// TIA Portal V17 program export: 3 tag tables, 41 data types, 3 data blocks, 7 code blocks (in call order from the OBs), 4 instance data blocks

VAR_GLOBAL   // PLC tag table "Constants"
END_VAR
VAR_GLOBAL CONSTANT   // user constants
   LASERCOMM_LDD_ARRAY_SIZE : Int := 100;   // Size of LDD Array Data Sizes. This is for Results, DDO and Weld Mask. Tied to the number of jobs in the LDD Sequence.
   LASERCOMM_NUMBER_OF_LASERS : Int := 1;   // Number of Lasers systems on Cell
   LASERCOMM_REF_PLANE : DInt := 12345;   // LDD Reference Plane Position
END_VAR

VAR_GLOBAL   // PLC tag table "Default tag table"
   Start_Seq AT %M0.0 : Bool;
   Rob_Reset_1 AT %M0.1 : Bool;
   Rob_Reset_2 AT %M0.2 : Bool;
   RA_CC_1 AT %M0.3 : Bool;
END_VAR
VAR_GLOBAL CONSTANT   // user constants
   GRP_JOB_NAME_SIZE : Int := 50;   // String site group and job name / String Größe Gruppen- und Jobnamen
   MAX_CNT_GRP_OVR_ENTRIES : DInt := 100;   // Maximum number of groups in the group overview / Maximale Anzahl Gruppen in der Gruppen-Übersicht
   MAX_CNT_MTN_OVR_ENTRIES : DInt := 150;   // Maximum number of motions in the motion overview / Maximale Anzahl Motions in der Motion-Übersicht
END_VAR

VAR_GLOBAL   // PLC tag table "Standard IO"
   iScanner1 AT %I0.0 : "Scanner_Inputs";
   oScanner1 AT %Q0.0 : "Scanner_Outputs";
   iLaser1 AT %I48.0 : "YLS_Inputs";
   oLaser1 AT %Q32.0 : "YLS_Outputs";
END_VAR

TYPE "typeAnalogSensorUniversalLimits"
// stored: IsFailsafeCompliant false
   STRUCT
      minPosition { ExternalAccessible := 'False'; ExternalVisible := 'False'; ExternalWritable := 'False'} : Array[1..8] of LReal;   // minimale Position / Minimum position
      maxPosition { ExternalAccessible := 'False'; ExternalVisible := 'False'; ExternalWritable := 'False'} : Array[1..8] of LReal;   // maximale Position / Maximum position
   END_STRUCT;
END_TYPE

TYPE "typeAnalogSensorUniversalPositions"
// stored: IsFailsafeCompliant false
   STRUCT
      inPosition { ExternalAccessible := 'False'; ExternalVisible := 'False'; ExternalWritable := 'False'} : Array[1..8] of Bool;   // in Position / In position
   END_STRUCT;
END_TYPE

TYPE "typeCaCgFg"
TITLE = Group / Gruppe
// Gruppe [V 01.09 | Kernel_V2]
// stored: IsFailsafeCompliant false
   STRUCT
      info { ExternalAccessible := 'False'; ExternalVisible := 'False'; ExternalWritable := 'False'} : Struct   // Info / Information
         "name" { ExternalAccessible := 'False'; ExternalVisible := 'False'; ExternalWritable := 'False'} : WString["GRP_JOB_NAME_SIZE"];   // Bezeichnung / Designation
         idString { ExternalAccessible := 'False'; ExternalVisible := 'False'; ExternalWritable := 'False'} : WString["GRP_JOB_NAME_SIZE"];   // ID-Bezeichnung als String (originaler Name des Gruppen-DB)
         groupType { ExternalAccessible := 'False'; ExternalVisible := 'False'; ExternalWritable := 'False'} : Int;   // Typ (1= CA | 2= CG | 3= FG) / Type (1 = CA | 2 = CG | 3 = FG)
         dbAdress { ExternalAccessible := 'False'; ExternalVisible := 'False'; ExternalWritable := 'False'} : DB_ANY;   // DB-Adresse der Gruppeschnittstelle (typeCaCgFg) / DB address of group interface (typeCaCgFg)
         panel { ExternalAccessible := 'False'; ExternalVisible := 'False'; ExternalWritable := 'False'} : Struct   // Panel
            assignment { ExternalAccessible := 'False'; ExternalVisible := 'False'; ExternalWritable := 'False'} : Int;   // Hmi Panel Zuweisung (Panel-Index aus HMI Lite) / HMI panel assignment (panel index from HMI Lite)
            memoryIndex { ExternalAccessible := 'False'; ExternalVisible := 'False'; ExternalWritable := 'False'} : Int;   // Speicherplatz Index Panel-Bild / Memory index panel screen
         END_STRUCT;
         parentGroup { ExternalAccessible := 'False'; ExternalVisible := 'False'; ExternalWritable := 'False'} : Struct   // Übergeordnete Gruppe / Superordinate group
            groupType { ExternalAccessible := 'False'; ExternalVisible := 'False'; ExternalWritable := 'False'} : Int;   // Übergeordnete Gruppe: Typ (1= CA | 2= CG | 3= FG) / Superordinate group: Type (1 = CA | 2 = CG | 3 = FG)
            "name" { ExternalAccessible := 'False'; ExternalVisible := 'False'; ExternalWritable := 'False'} : WString["GRP_JOB_NAME_SIZE"];   // Übergeordnete Gruppe: Bezeichnung / Superordinate group: Designation
            dbAdress { ExternalAccessible := 'False'; ExternalVisible := 'False'; ExternalWritable := 'False'} : DB_ANY;   // Übergeordnete Gruppe: DB-Adresse der Gruppeschnittstelle (typeCaCgFg) / Superordinate group: DB address of group interface (typeCaCgFg)
         END_STRUCT;
         groupOvrv { ExternalAccessible := 'False'; ExternalVisible := 'False'; ExternalWritable := 'False'} : Struct   // Gruppenübersichtstabelle: ... / Group overview table: ...
            groupOvrvAdress { ExternalAccessible := 'False'; ExternalVisible := 'False'; ExternalWritable := 'False'} : DB_ANY;   // Gruppenübersichtstabelle: Adresse auf Gruppenübersichts-DB (typeGroupOvrvList) / Group overview table: address on group overview DB (typeGroupOvrvList)
            listedIndex { ExternalAccessible := 'False'; ExternalVisible := 'False'; ExternalWritable := 'False'} : DInt := -1;   // Gruppenübersichtstabelle: Index der Gruppe im Gruppenübersichts-DB / Group overview table: group index in group overview DB
         END_STRUCT;
         motionOvrv { ExternalAccessible := 'False'; ExternalVisible := 'False'; ExternalWritable := 'False'} : Struct   // Motion-Übersichtstabelle: ... (Wird nur in einer FG beschrieben!) / Motion overview table: ... (only described in one FG!)
            enabled { ExternalAccessible := 'False'; ExternalVisible := 'False'; ExternalWritable := 'False'} : Bool;   // Motion-Übersichtstabelle: Freigeschaltet / Motion overview: activated
            motionOvrvAdress { ExternalAccessible := 'False'; ExternalVisible := 'False'; ExternalWritable := 'False'} : DB_ANY;   // Motion-Übersichtstabelle: Adresse auf Motion-Übersichts-DB (typeMotionOvrvList) / Motion overview table: address on motion overview DB (typeMotionOvrvList)
         END_STRUCT;
      END_STRUCT;
      groupModes { ExternalAccessible := 'False'; ExternalVisible := 'False'; ExternalWritable := 'False'} : Struct   // Gruppen Modus / Station mode <ToBeDone: determine symbol> / Group mode
         activation { ExternalAccessible := 'False'; ExternalVisible := 'False'; ExternalWritable := 'False'} : Struct   // Gruppen-Aktivierung / Group activation
            deactivate { ExternalAccessible := 'False'; ExternalVisible := 'False'; ExternalWritable := 'False'} : Bool;   // Gruppe deaktivieren (S) / Deactivate group (S)
            activate { ExternalAccessible := 'False'; ExternalVisible := 'False'; ExternalWritable := 'False'} : Bool;   // Gruppe aktivieren (S) / Activate group (S)
            isDeactived { ExternalAccessible := 'False'; ExternalVisible := 'False'; ExternalWritable := 'False'} : Bool;   // Gruppe ist deaktiviert / Group deactivated
         END_STRUCT;
         interlinkedMode { ExternalAccessible := 'False'; ExternalVisible := 'False'; ExternalWritable := 'False'} : Struct   // Verketteter Betrieb / Interlinked mode
            select { ExternalAccessible := 'False'; ExternalVisible := 'False'; ExternalWritable := 'False'} : Bool;   // Anwahl verketteter Betrieb (S) / Selection of interlinked mode (S)
            deselect { ExternalAccessible := 'False'; ExternalVisible := 'False'; ExternalWritable := 'False'} : Bool;   // Abwahl verketteter Betrieb (S) / Deselection of interlinked mode (S)
            isActive { ExternalAccessible := 'False'; ExternalVisible := 'False'; ExternalWritable := 'False'} : Bool;   // Verketteter Betrieb ist aktiv / Interlinked mode active
         END_STRUCT;
      END_STRUCT;
      enable { ExternalAccessible := 'False'; ExternalVisible := 'False'; ExternalWritable := 'False'} : Struct   // Freigaben / Enables
         hardware { ExternalAccessible := 'False'; ExternalVisible := 'False'; ExternalWritable := 'False'} : Bool;   // Freigabe Hardware betriebsbereit / Enable hardware ready for operation
         safety { ExternalAccessible := 'False'; ExternalVisible := 'False'; ExternalWritable := 'False'} : Bool;   // Freigabe Schutzbereich Bewegungsfreigabe / Enable guarded area movement enable
         enterSafeArea { ExternalAccessible := 'False'; ExternalVisible := 'False'; ExternalWritable := 'False'} : Struct   // Freigabe Zugang Schutzbereich / Enable for access guarded area
            isEnabled { ExternalAccessible := 'False'; ExternalVisible := 'False'; ExternalWritable := 'False'} : Bool;   // Zugang zum Schutzbereich ist freigegeben / Access to guarded area enabled
            disable { ExternalAccessible := 'False'; ExternalVisible := 'False'; ExternalWritable := 'False'} : Bool;   // Freigabe Zugnag Schutzbereich sperren (S) / Enable for lock access guarded area (S)
            disableSelected { ExternalAccessible := 'False'; ExternalVisible := 'False'; ExternalWritable := 'False'} : Bool;   // Freigabe Zugnag Schutzbereich sperren ist Angewählt / Enable for lock access guarded area is selected
            request { ExternalAccessible := 'False'; ExternalVisible := 'False'; ExternalWritable := 'False'} : Bool;   // Freigabe Zugang Schutzbereich anfordern (S) / Request enable for access guarded area (S)
            isRequested { ExternalAccessible := 'False'; ExternalVisible := 'False'; ExternalWritable := 'False'} : Bool;   // Freigabe Zugang Schutzbereich ist anfordert / Enable for access guarded area is requested
            operatorGuidance { ExternalAccessible := 'False'; ExternalVisible := 'False'; ExternalWritable := 'False'} : Struct   // Freigabe Zugang Schutzbereich Bedienerführung / Operator guidance guarded area access enable
               select { ExternalAccessible := 'False'; ExternalVisible := 'False'; ExternalWritable := 'False'} : Bool;   // Freigabe Zugang Schutzbereich Bedienerführung Anwahl (S) / Enable for access guarded area operator guidance selection (S)
               isSelected { ExternalAccessible := 'False'; ExternalVisible := 'False'; ExternalWritable := 'False'} : Bool;   // Freigabe Zugang Schutzbereich Bedienerführung angewählt / Operator guidance guarded area access enable selected
            END_STRUCT;
         END_STRUCT;
      END_STRUCT;
      baseFunction { ExternalAccessible := 'False'; ExternalVisible := 'False'; ExternalWritable := 'False'} : Struct   // Grundfunktionen / Basic functions
         homePos { ExternalAccessible := 'False'; ExternalVisible := 'False'; ExternalWritable := 'False'} : Struct   // Grundfunktion: Grundstellung / Basic function: home position
            select { ExternalAccessible := 'False'; ExternalVisible := 'False'; ExternalWritable := 'False'} : Bool;   // Grundfunktion: Anwahl "Zur Grundstellung" (S) / Basic function: selection "To home position" (S)
            isSelected { ExternalAccessible := 'False'; ExternalVisible := 'False'; ExternalWritable := 'False'} : Bool;   // Grundfunktion: "Zur Grundstellung" angewählt / Basic function: "To home position" selected
            isPending { ExternalAccessible := 'False'; ExternalVisible := 'False'; ExternalWritable := 'False'} : Bool;   // Grundfunktion: "Zur Grundstellung" steht an (aktiv oder gestoppt) / Basic function: "To home position" pending (active or stopped)
            inExecution { ExternalAccessible := 'False'; ExternalVisible := 'False'; ExternalWritable := 'False'} : Bool;   // Grundfunktion: "Zur Grundstellung" aktiv / Basic function: "To home position" active
            inExecutionPulse { ExternalAccessible := 'False'; ExternalVisible := 'False'; ExternalWritable := 'False'} : Bool;   // Grundfunktion: "Zur Grundstellung" aktiv Impuls / To home position active impulse / Basic function: "To home pos." active impulse
            inState { ExternalAccessible := 'False'; ExternalVisible := 'False'; ExternalWritable := 'False'} : Bool;   // Grundfunktion: In Grundstellung / Basic function: in home position
            display { ExternalAccessible := 'False'; ExternalVisible := 'False'; ExternalWritable := 'False'} : Bool;   // Grundfunktion: Grundstellung Anzeige / Basic function: home position display
            operatorGuidance { ExternalAccessible := 'False'; ExternalVisible := 'False'; ExternalWritable := 'False'} : Struct   // Grundfunktion: Bedienerfürhung / Basic function: Operator guidance
               select { ExternalAccessible := 'False'; ExternalVisible := 'False'; ExternalWritable := 'False'} : Bool;   // Grundfunktion: Bedienerfürhung Anwahl (S) / Basic function: Operator guidance selection (S)
               isSelected { ExternalAccessible := 'False'; ExternalVisible := 'False'; ExternalWritable := 'False'} : Bool;   // Grundfunktion: Bedienerfürhung Angewählt / Basic function: Operator guidance selected
            END_STRUCT;
         END_STRUCT;
         start { ExternalAccessible := 'False'; ExternalVisible := 'False'; ExternalWritable := 'False'} : Struct   // Grundfunktion: Start / Basic function: start
            select { ExternalAccessible := 'False'; ExternalVisible := 'False'; ExternalWritable := 'False'} : Bool;   // Grundfunktion: Anwah Startl (S) / Basic function: selection start (S)
            isSelected { ExternalAccessible := 'False'; ExternalVisible := 'False'; ExternalWritable := 'False'} : Bool;   // Grundfunktion: Start angewählt / Basic function: start selected
            isPending { ExternalAccessible := 'False'; ExternalVisible := 'False'; ExternalWritable := 'False'} : Bool;   // Grundfunktion: Start steht an (aktiv oder gestoppt) / Basic function: Start pending (active or stopped)
            inExecution { ExternalAccessible := 'False'; ExternalVisible := 'False'; ExternalWritable := 'False'} : Bool;   // Grundfunktion: Start ist aktiv / Basic function: start active
            inExecutionPulse { ExternalAccessible := 'False'; ExternalVisible := 'False'; ExternalWritable := 'False'} : Bool;   // Grundfunktion: Start ist aktiv Impuls / Basic function: start active pulse
            inState { ExternalAccessible := 'False'; ExternalVisible := 'False'; ExternalWritable := 'False'} : Bool;   // Grundfunktion: Gestartet / Basic function: started
            display { ExternalAccessible := 'False'; ExternalVisible := 'False'; ExternalWritable := 'False'} : Bool;   // Grundfunktion: Start Anzeige / Basic function: start display
            operatorGuidance { ExternalAccessible := 'False'; ExternalVisible := 'False'; ExternalWritable := 'False'} : Struct   // Grundfunktion: Start Bedienerführung / Basic function: start operator guidance start
               select { ExternalAccessible := 'False'; ExternalVisible := 'False'; ExternalWritable := 'False'} : Bool;   // Grundfunktion: Start Bedienerführung Anwahl (S) / Basic function: start operator guidance selection (S)
               isSelected { ExternalAccessible := 'False'; ExternalVisible := 'False'; ExternalWritable := 'False'} : Bool;   // Grundfunktion: Start Bedienerführung Angewählt / Basic function: Operator guidance start selected
            END_STRUCT;
         END_STRUCT;
         stop { ExternalAccessible := 'False'; ExternalVisible := 'False'; ExternalWritable := 'False'} : Struct   // Grundfunktion: Stop / Basic function: stop
            select { ExternalAccessible := 'False'; ExternalVisible := 'False'; ExternalWritable := 'False'} : Bool;   // Grundfunktion: Anwahl Stop generell (S) (wählt Stop für alle Auslöser an) / Basic function: selection stop (S)
            selectBy { ExternalAccessible := 'False'; ExternalVisible := 'False'; ExternalWritable := 'False'} : Struct   // Grundfunktion: Anwahl Stop nach Auslöser ...
               manual { ExternalAccessible := 'False'; ExternalVisible := 'False'; ExternalWritable := 'False'} : Bool;   // Grundfunktion: Anwahl Stop durch Bedienung (S)
               fault { ExternalAccessible := 'False'; ExternalVisible := 'False'; ExternalWritable := 'False'} : Bool;   // Grundfunktion: Anwahl Stop durch Störung (S)
               system { ExternalAccessible := 'False'; ExternalVisible := 'False'; ExternalWritable := 'False'} : Bool;   // Grundfunktion: Anwahl Stop durch System (S)
            END_STRUCT;
            isSelected { ExternalAccessible := 'False'; ExternalVisible := 'False'; ExternalWritable := 'False'} : Bool;   // Grundfunktion: Stop angewählt generell (alle Auslöser) / Basic function: stop selected
            isSelectedBy { ExternalAccessible := 'False'; ExternalVisible := 'False'; ExternalWritable := 'False'} : Struct   // Grundfunktion: Stop angewählt nach Auslöser ...
               manual { ExternalAccessible := 'False'; ExternalVisible := 'False'; ExternalWritable := 'False'} : Bool;   // Grundfunktion: Stop angewählt durch Bedienung
               fault { ExternalAccessible := 'False'; ExternalVisible := 'False'; ExternalWritable := 'False'} : Bool;   // Grundfunktion: Stop angewählt durch Störung
               system { ExternalAccessible := 'False'; ExternalVisible := 'False'; ExternalWritable := 'False'} : Bool;   // Grundfunktion: Stop angewählt durch System
            END_STRUCT;
            isPending { ExternalAccessible := 'False'; ExternalVisible := 'False'; ExternalWritable := 'False'} : Bool;   // Grundfunktion: Stop steht an / Basic function: Stop pending
            inExecution { ExternalAccessible := 'False'; ExternalVisible := 'False'; ExternalWritable := 'False'} : Bool;   // Grundfunktion: Stop ist aktiv / Basic function: stop active
            inState { ExternalAccessible := 'False'; ExternalVisible := 'False'; ExternalWritable := 'False'} : Bool;   // Grundfunktion: Gestoppt / Basic function: stopped
            display { ExternalAccessible := 'False'; ExternalVisible := 'False'; ExternalWritable := 'False'} : Bool;   // Grundfunktion: Stop Anzeige / Basic function: stop display
            operatorGuidance { ExternalAccessible := 'False'; ExternalVisible := 'False'; ExternalWritable := 'False'} : Struct   // Grundfunktion: Stop Bedienerfürhung / Basic function: Operator guidance stop
               select { ExternalAccessible := 'False'; ExternalVisible := 'False'; ExternalWritable := 'False'} : Bool;   // Grundfunktion: Stop Bedienerfürhung Anwahl (S) / Basic function: Operator guidance stop selection (S)
               isSelected { ExternalAccessible := 'False'; ExternalVisible := 'False'; ExternalWritable := 'False'} : Bool;   // Grundfunktion: Stop Bedienerfürhung Angewählt / Basic function: Operator guidance stop selected
            END_STRUCT;
         END_STRUCT;
         reset { ExternalAccessible := 'False'; ExternalVisible := 'False'; ExternalWritable := 'False'} : Struct   // Grundfunktion: Reset / Basic function: reset
            select { ExternalAccessible := 'False'; ExternalVisible := 'False'; ExternalWritable := 'False'} : Bool;   // Grundfunktion: Anwahl Reset (S) / Basic function: selection reset (S)
            isSelected { ExternalAccessible := 'False'; ExternalVisible := 'False'; ExternalWritable := 'False'} : Bool;   // Grundfunktion: Reset angewählt / Basic function: reset selected
            isPending { ExternalAccessible := 'False'; ExternalVisible := 'False'; ExternalWritable := 'False'} : Bool;   // Grundfunktion: Reset steht an / Basic function: Reset pending
            inExecution { ExternalAccessible := 'False'; ExternalVisible := 'False'; ExternalWritable := 'False'} : Bool;   // Grundfunktion: Reset ist aktiv / Basic function: reset is active
            inState { ExternalAccessible := 'False'; ExternalVisible := 'False'; ExternalWritable := 'False'} : Bool;   // Grundfunktion: Im Reset / Basic function: in reset
            display { ExternalAccessible := 'False'; ExternalVisible := 'False'; ExternalWritable := 'False'} : Bool;   // Grundfunktion: Reset Anzeige / Basic function: reset display
            operatorGuidance { ExternalAccessible := 'False'; ExternalVisible := 'False'; ExternalWritable := 'False'} : Struct   // Grundfunktion: Reset Bedienerführung / Basic function: Operator guidance reset
               select { ExternalAccessible := 'False'; ExternalVisible := 'False'; ExternalWritable := 'False'} : Bool;   // Grundfunktion: Reset Bedienerführung Anwahl (S) / Basic function: reset operator guidance selection (S)
               isSelected { ExternalAccessible := 'False'; ExternalVisible := 'False'; ExternalWritable := 'False'} : Bool;   // Grundfunktion: Reset Bedienerführung angewählt / Basic function: Operator guidance reset selected
            END_STRUCT;
         END_STRUCT;
         stopCycleEnd { ExternalAccessible := 'False'; ExternalVisible := 'False'; ExternalWritable := 'False'} : Struct   // Grundfunktion: "Halt nach Taktende" / Basic function: "Stop at end of cycle"
            select { ExternalAccessible := 'False'; ExternalVisible := 'False'; ExternalWritable := 'False'} : Bool;   // Grundfunktion: Anwahl "Halt nach Taktende" (S) / Basic function: selection "Stop at end of cycle" (S)
            isSelected { ExternalAccessible := 'False'; ExternalVisible := 'False'; ExternalWritable := 'False'} : Bool;   // Grundfunktion: "Halt nach Taktende" angewählt / Basic function: "Stop at end of cycle" selected
            isPending { ExternalAccessible := 'False'; ExternalVisible := 'False'; ExternalWritable := 'False'} : Bool;   // Grundfunktion: "Halt nach Taktende" steht an / Basic function: "Stop at end of cycle" pending
            inExecution { ExternalAccessible := 'False'; ExternalVisible := 'False'; ExternalWritable := 'False'} : Bool;   // Grundfunktion: "Halt nach Taktende" aktiv / Basic function: "Stop at end of cycle" active
            inState { ExternalAccessible := 'False'; ExternalVisible := 'False'; ExternalWritable := 'False'} : Bool;   // Grundfunktion: "Halt nach Taktende" erreicht / Basic function: "Stop at end of cycle" reached
            display { ExternalAccessible := 'False'; ExternalVisible := 'False'; ExternalWritable := 'False'} : Bool;   // Grundfunktion: "Halt nach Taktende" Anzeige / Basic function: "Stop at end of cycle" display
            operatorGuidance { ExternalAccessible := 'False'; ExternalVisible := 'False'; ExternalWritable := 'False'} : Struct   // Grundfunktion: "Halt nach Taktende" Bedienerführung / Basic function: "Stop at end of cycle" operator guidance
               select { ExternalAccessible := 'False'; ExternalVisible := 'False'; ExternalWritable := 'False'} : Bool;   // Grundfunktion: "Halt nach Taktende" Bedienerführung Anwahl (S) / Basic function: "Stop at end of cycle" operator guidance selection (S)
               isSelected { ExternalAccessible := 'False'; ExternalVisible := 'False'; ExternalWritable := 'False'} : Bool;   // Grundfunktion: "Halt nach Taktende" Bedienerführung angewählt / Basic function: "Stop at end of cycle" operator guidance selected
            END_STRUCT;
         END_STRUCT;
         singleCycleStep { ExternalAccessible := 'False'; ExternalVisible := 'False'; ExternalWritable := 'False'} : Struct   // Grundfunktionen Einzelbetrieb/Einzelschritt / Basic functions single cycle/single step
            jobSelected { ExternalAccessible := 'False'; ExternalVisible := 'False'; ExternalWritable := 'False'} : Bool;   // Grundfunktionen Einzelbetrieb/Einzelschritt: Auftrag angewählt / Basic functions single cycle/single step: job selected
            homePosStep { ExternalAccessible := 'False'; ExternalVisible := 'False'; ExternalWritable := 'False'} : Struct   // Grundfunktion Grundstellung Einzelschritt / Basic function home position single-step
               jobSelected { ExternalAccessible := 'False'; ExternalVisible := 'False'; ExternalWritable := 'False'} : Bool;   // Grundfunktion Grundstellung Einzelschritt: Auftrag angewählt / Basic function home position single-step: Job selected
               active { ExternalAccessible := 'False'; ExternalVisible := 'False'; ExternalWritable := 'False'} : Bool;   // Grundfunktion Grundstellung Einzelschritt: Aktiv / Basic function home position single-step: Active
            END_STRUCT;
         END_STRUCT;
         startOrToHomePosActive { ExternalAccessible := 'False'; ExternalVisible := 'False'; ExternalWritable := 'False'} : Bool;   // Start oder "Zur Grundstellung" aktiv / Start or "To home position" active
         stoppedOrInReset { ExternalAccessible := 'False'; ExternalVisible := 'False'; ExternalWritable := 'False'} : Bool;   // Gestoppt oder im Reset / Stopped or in reset
      END_STRUCT;
      operatingMode { ExternalAccessible := 'False'; ExternalVisible := 'False'; ExternalWritable := 'False'} : Struct   // Funktionsarten / Operating modes / Function types
         automatic { ExternalAccessible := 'False'; ExternalVisible := 'False'; ExternalWritable := 'False'} : Struct   // Funktionsart Automatik / Automatic operating mode / Function type automatic
            select { ExternalAccessible := 'False'; ExternalVisible := 'False'; ExternalWritable := 'False'} : Bool;   // Funktionsart Automatik Anwahl (S) / Automatic mode selection (S)
            isActive { ExternalAccessible := 'False'; ExternalVisible := 'False'; ExternalWritable := 'False'} : Bool;   // Funktionsart Automatik aktiv / Automatic mode active
            operatorGuidance { ExternalAccessible := 'False'; ExternalVisible := 'False'; ExternalWritable := 'False'} : Struct   // Funktionsart Automatik Bedienerführung / Automatic mode operator guidance
               select { ExternalAccessible := 'False'; ExternalVisible := 'False'; ExternalWritable := 'False'} : Bool;   // Funktionsart Automatik Bedienerführung Anwahl (S) / Automatic mode operator guidance selection (S)
               isSelected { ExternalAccessible := 'False'; ExternalVisible := 'False'; ExternalWritable := 'False'} : Bool;   // Funktionsart Automatik Bedienerführung angewählt / Automatic mode operator guidance selected
            END_STRUCT;
         END_STRUCT;
         singleCycle { ExternalAccessible := 'False'; ExternalVisible := 'False'; ExternalWritable := 'False'} : Struct   // Funktionsart Einzelbetrieb / Semi-automatic mode / Function type single mode
            select { ExternalAccessible := 'False'; ExternalVisible := 'False'; ExternalWritable := 'False'} : Bool;   // Funktionsart Einzelbetrieb Anwahl (S) / Single cycle mode selection (S) / Single operation mode selection (S)
            isActive { ExternalAccessible := 'False'; ExternalVisible := 'False'; ExternalWritable := 'False'} : Bool;   // Funktionsart Einzelbetrieb aktiv / Operating mode single cycle active / Single operation mode active
            operatorGuidance { ExternalAccessible := 'False'; ExternalVisible := 'False'; ExternalWritable := 'False'} : Struct   // Funktionsart Einzelbetrieb Bedienerführung / Single operation mode operator guidance
               select { ExternalAccessible := 'False'; ExternalVisible := 'False'; ExternalWritable := 'False'} : Bool;   // Funktionsart Einzelbetrieb Bedienerführung Anwahl (S) / Single operation mode operator guidance selection (S)
               isSelected { ExternalAccessible := 'False'; ExternalVisible := 'False'; ExternalWritable := 'False'} : Bool;   // Funktionsart Einzelbetrieb Bedienerführung angewählt / Single operation mode operator guidance selected
            END_STRUCT;
         END_STRUCT;
         singleStep { ExternalAccessible := 'False'; ExternalVisible := 'False'; ExternalWritable := 'False'} : Struct   // Funktionsart Einzelschritt / Operating mode Single step / Function type single step
            select { ExternalAccessible := 'False'; ExternalVisible := 'False'; ExternalWritable := 'False'} : Bool;   // Funktionsart Einzelschritt Anwahl (S) / Single step mode selection (S) / Single-step mode selection (S)
            isActive { ExternalAccessible := 'False'; ExternalVisible := 'False'; ExternalWritable := 'False'} : Bool;   // Funktionsart Einzelschritt aktiv / Single step mode active / Single-step mode active
            operatorGuidance { ExternalAccessible := 'False'; ExternalVisible := 'False'; ExternalWritable := 'False'} : Struct   // Funktionsart Einzelschritt Bedienerfürhung / Single-step mode operator guidance
               select { ExternalAccessible := 'False'; ExternalVisible := 'False'; ExternalWritable := 'False'} : Bool;   // Funktionsart Einzelschritt Bedienerfürhung Anwahl (S) / Single-step mode operator guidance selection (S)
               isSelected { ExternalAccessible := 'False'; ExternalVisible := 'False'; ExternalWritable := 'False'} : Bool;   // Funktionsart Einzelschritt Bedienerfürhung angewählt / Single-step mode operator guidance selected
            END_STRUCT;
         END_STRUCT;
         manual { ExternalAccessible := 'False'; ExternalVisible := 'False'; ExternalWritable := 'False'} : Struct   // Funktionsart Einrichten / setup mode / Function start setup mode
            select { ExternalAccessible := 'False'; ExternalVisible := 'False'; ExternalWritable := 'False'} : Bool;   // Funktionsart Einrichten Anwahl (S) / Setup mode selection (S)
            isActive { ExternalAccessible := 'False'; ExternalVisible := 'False'; ExternalWritable := 'False'} : Bool;   // Funktionsart Einrichten aktiv / Setup Mode Active / Setup mode active
            operatorGuidance { ExternalAccessible := 'False'; ExternalVisible := 'False'; ExternalWritable := 'False'} : Struct   // Funktionsart Einrichten Bedienerführung / Setup mode operator guidance
               select { ExternalAccessible := 'False'; ExternalVisible := 'False'; ExternalWritable := 'False'} : Bool;   // Funktionsart Einrichten Bedienerführung Anwahl (S) / Setup mode operator guidance selection (S)
               isSelected { ExternalAccessible := 'False'; ExternalVisible := 'False'; ExternalWritable := 'False'} : Bool;   // Funktionsart Einrichten Bedienerführung angewählt / Setup mode operator guidance selected
            END_STRUCT;
         END_STRUCT;
      END_STRUCT;
      cycleType { ExternalAccessible := 'False'; ExternalVisible := 'False'; ExternalWritable := 'False'} : Struct   // Taktarten / Cycle types
         warmUp { ExternalAccessible := 'False'; ExternalVisible := 'False'; ExternalWritable := 'False'} : Struct   // Taktart Warmfahren / Cycle type warm-up
            select { ExternalAccessible := 'False'; ExternalVisible := 'False'; ExternalWritable := 'False'} : Bool;   // Taktart Warmfahren: Anwahl (S) / Cycle type warm-up: selection (S)
            deselect { ExternalAccessible := 'False'; ExternalVisible := 'False'; ExternalWritable := 'False'} : Bool;   // Taktart Warmfahren: Abwahl (S) / Cycle type warm-up: deselection (S)
            isActive { ExternalAccessible := 'False'; ExternalVisible := 'False'; ExternalWritable := 'False'} : Bool;   // Taktart Warmfahren: Aktiv / Cycle type warm-up: active
            operatorGuidance { ExternalAccessible := 'False'; ExternalVisible := 'False'; ExternalWritable := 'False'} : Struct   // Taktart Warmfahren: Bedienerführung / Warm-up cycle type: Operator guidance
               select { ExternalAccessible := 'False'; ExternalVisible := 'False'; ExternalWritable := 'False'} : Bool;   // Taktart Warmfahren: Bedienerführung Anwahl (S) / Cycle type warm-up: operator guidance selection (S)
               isSelected { ExternalAccessible := 'False'; ExternalVisible := 'False'; ExternalWritable := 'False'} : Bool;   // Taktart Warmfahren: Bedienerführung angewählt / Warm-up cycle type: Operator guidance selected
            END_STRUCT;
         END_STRUCT;
         runOut { ExternalAccessible := 'False'; ExternalVisible := 'False'; ExternalWritable := 'False'} : Struct   // Taktart Leerfahren / Cycle type runout mode
            select { ExternalAccessible := 'False'; ExternalVisible := 'False'; ExternalWritable := 'False'} : Bool;   // Taktart Leerfahren: Anwahl (S) / Cycle type runout mode: selection (S)
            deselect { ExternalAccessible := 'False'; ExternalVisible := 'False'; ExternalWritable := 'False'} : Bool;   // Taktart Leerfahren: Abwahl (S) / Cycle type runout mode: deselection (S)
            isActive { ExternalAccessible := 'False'; ExternalVisible := 'False'; ExternalWritable := 'False'} : Bool;   // Taktart Leerfahren: Aktiv / Cycle type runout mode: active
            operatorGuidance { ExternalAccessible := 'False'; ExternalVisible := 'False'; ExternalWritable := 'False'} : Struct   // Taktart Leerfahren: Bedienerführung / Runout mode cycle type: Operator guidance
               select { ExternalAccessible := 'False'; ExternalVisible := 'False'; ExternalWritable := 'False'} : Bool;   // Taktart Leerfahren: Bedienerführung Anwahl (S) / Cycle type runout mode: oeprator guidance selection (S)
               isSelected { ExternalAccessible := 'False'; ExternalVisible := 'False'; ExternalWritable := 'False'} : Bool;   // Taktart Leerfahren: Bedienerführung angewählt / Runout mode cycle type: Operator guidance selected
            END_STRUCT;
            selectedByUpperLevel { ExternalAccessible := 'False'; ExternalVisible := 'False'; ExternalWritable := 'False'} : Bool;   // Taktart Leerfahren: Durch übergeordnete Ebene anewählt (CA / CG) / Runout mode was selected in other level / Runout mode cycle type: Selected by higher level (CA / CG)
         END_STRUCT;
         withoutPart { ExternalAccessible := 'False'; ExternalVisible := 'False'; ExternalWritable := 'False'} : Struct   // Taktart "Fahren ohne Werkstück" / Cycle type <Traverse without part>
            select { ExternalAccessible := 'False'; ExternalVisible := 'False'; ExternalWritable := 'False'} : Bool;   // Taktart "Fahren ohne Werkstück": Anwahl (S) / Cycle type "Traverse without part": selection (S)
            deselect { ExternalAccessible := 'False'; ExternalVisible := 'False'; ExternalWritable := 'False'} : Bool;   // Taktart "Fahren ohne Werkstück": Abwahl (S) / Cycle type "Traverse without part": deselection (S)
            isActive { ExternalAccessible := 'False'; ExternalVisible := 'False'; ExternalWritable := 'False'} : Bool;   // Taktart "Fahren ohne Werkstück": Aktiv / Cycle type "Traverse without part": active
            operatorGuidance { ExternalAccessible := 'False'; ExternalVisible := 'False'; ExternalWritable := 'False'} : Struct   // Taktart "Fahren ohne Werkstück": Bedienerführung / Cycle type "Traverse without part": Operator guidance
               select { ExternalAccessible := 'False'; ExternalVisible := 'False'; ExternalWritable := 'False'} : Bool;   // Taktart "Fahren ohne Werkstück": Bedienerführung Anwahl (S) / Cycle type "Traverse without part": operator guidance selection (S)
               isSelected { ExternalAccessible := 'False'; ExternalVisible := 'False'; ExternalWritable := 'False'} : Bool;   // Taktart "Fahren ohne Werkstück": Bedienerführung angewählt / Cycle type "Traverse without part": Operator guidance selected
            END_STRUCT;
         END_STRUCT;
         userDefined1 { ExternalAccessible := 'False'; ExternalVisible := 'False'; ExternalWritable := 'False'} : Struct   // Taktart Benutzerdefiniert 1 / User-defined cycle type 1
            select { ExternalAccessible := 'False'; ExternalVisible := 'False'; ExternalWritable := 'False'} : Bool;   // Taktart Benutzerdefiniert 1: Anwahl (S) / User-defined cycle type 1: Selection (S)
            deselect { ExternalAccessible := 'False'; ExternalVisible := 'False'; ExternalWritable := 'False'} : Bool;   // Taktart Benutzerdefiniert 1: Abwahl (S) / User-defined cycle type 1: Deselection (S)
            isActive { ExternalAccessible := 'False'; ExternalVisible := 'False'; ExternalWritable := 'False'} : Bool;   // Taktart Benutzerdefiniert 1: Aktiv / User-defined cycle type 1: Active
            operatorGuidance { ExternalAccessible := 'False'; ExternalVisible := 'False'; ExternalWritable := 'False'} : Struct   // Taktart Benutzerdefiniert 1: Bedienerführung / User-defined cycle type 1: Operator guidance
               select { ExternalAccessible := 'False'; ExternalVisible := 'False'; ExternalWritable := 'False'} : Bool;   // Taktart Benutzerdefiniert 1: Bedienerführung Anwahl (S) / User-defined cycle type 1: Operator guidance selection (S)
               isSelected { ExternalAccessible := 'False'; ExternalVisible := 'False'; ExternalWritable := 'False'} : Bool;   // Taktart Benutzerdefiniert 1: Bedienerführung angewählt / User-defined cycle type 1: Operator guidance selected
            END_STRUCT;
         END_STRUCT;
         userDefined2 { ExternalAccessible := 'False'; ExternalVisible := 'False'; ExternalWritable := 'False'} : Struct   // Taktart Benutzerdefiniert 2 / User-defined cycle type 2
            select { ExternalAccessible := 'False'; ExternalVisible := 'False'; ExternalWritable := 'False'} : Bool;   // Taktart Benutzerdefiniert 2: Anwahl (S) / User-defined cycle type 2: Selection (S)
            deselect { ExternalAccessible := 'False'; ExternalVisible := 'False'; ExternalWritable := 'False'} : Bool;   // Taktart Benutzerdefiniert 2: Abwahl (S) / User-defined cycle type 2: Deselection (S)
            isActive { ExternalAccessible := 'False'; ExternalVisible := 'False'; ExternalWritable := 'False'} : Bool;   // Taktart Benutzerdefiniert 2: Aktiv / User-defined cycle type 2: Active
            operatorGuidance { ExternalAccessible := 'False'; ExternalVisible := 'False'; ExternalWritable := 'False'} : Struct   // Taktart Benutzerdefiniert 2: Bedienerführung / User-defined cycle type 2: Operator guidance
               select { ExternalAccessible := 'False'; ExternalVisible := 'False'; ExternalWritable := 'False'} : Bool;   // Taktart Benutzerdefiniert 2: Bedienerführung Anwahl (S) / User-defined cycle type 2: Operator guidance selection (S)
               isSelected { ExternalAccessible := 'False'; ExternalVisible := 'False'; ExternalWritable := 'False'} : Bool;   // Taktart Benutzerdefiniert 2: Bedienerführung angewählt / User-defined cycle type 2: Operator guidance selected
            END_STRUCT;
         END_STRUCT;
      END_STRUCT;
      specialSignal { ExternalAccessible := 'False'; ExternalVisible := 'False'; ExternalWritable := 'False'} : Struct   // Sonder-Signale / Special signals
         userLevel { ExternalAccessible := 'False'; ExternalVisible := 'False'; ExternalWritable := 'False'} : "typeUserLevel";   // Benutzerlevel / User level
         isEmpty { ExternalAccessible := 'False'; ExternalVisible := 'False'; ExternalWritable := 'False'} : Bool;   // Ist leer / Is empty
         serviceMode { ExternalAccessible := 'False'; ExternalVisible := 'False'; ExternalWritable := 'False'} : Struct   // Servicemodus / Service mode
            select { ExternalAccessible := 'False'; ExternalVisible := 'False'; ExternalWritable := 'False'} : Bool;   // Servicemodus: Anwahl (S) / Service mode: selection (S)
            deselect { ExternalAccessible := 'False'; ExternalVisible := 'False'; ExternalWritable := 'False'} : Bool;   // Servicemodus: Abwahl (S) / Service mode: deselection (S)
            isActive { ExternalAccessible := 'False'; ExternalVisible := 'False'; ExternalWritable := 'False'} : Bool;   // Servicemodus: Aktiv / Service mode: active
            operatorGuidance { ExternalAccessible := 'False'; ExternalVisible := 'False'; ExternalWritable := 'False'} : Struct   // Servicemodus: Bedienerführung / Service mode: Operator guidance
               select { ExternalAccessible := 'False'; ExternalVisible := 'False'; ExternalWritable := 'False'} : Bool;   // Servicemodus: Bedienerführung Anwahl (S) / Service mode: Operator guidance selection (S)
               isSelected { ExternalAccessible := 'False'; ExternalVisible := 'False'; ExternalWritable := 'False'} : Bool;   // Servicemodus: Bedienerführung angewählt / Service mode: Operator guidance selected
            END_STRUCT;
         END_STRUCT;
         userDefined1 { ExternalAccessible := 'False'; ExternalVisible := 'False'; ExternalWritable := 'False'} : Struct   // Service Benutzerdefiniert 1 / User-defined service 1
            select { ExternalAccessible := 'False'; ExternalVisible := 'False'; ExternalWritable := 'False'} : Bool;   // Service Benutzerdefiniert 1: Anwahl (S) / User-defined service 1: Selection (S)
            deselect { ExternalAccessible := 'False'; ExternalVisible := 'False'; ExternalWritable := 'False'} : Bool;   // Service Benutzerdefiniert 1: Abwahl (S) / User-defined service 1: Deselection (S)
            isActive { ExternalAccessible := 'False'; ExternalVisible := 'False'; ExternalWritable := 'False'} : Bool;   // Service Benutzerdefiniert 1: Aktiv / User-defined service 1: Active
            operatorGuidance { ExternalAccessible := 'False'; ExternalVisible := 'False'; ExternalWritable := 'False'} : Struct   // Service Benutzerdefiniert 1: Bedienerführung / User-defined service 1: Operator guidance
               select { ExternalAccessible := 'False'; ExternalVisible := 'False'; ExternalWritable := 'False'} : Bool;   // Service Benutzerdefiniert 1: Bedienerführung Anwahl (S) / User-defined service 1: Operator guidance selection (S)
               isSelected { ExternalAccessible := 'False'; ExternalVisible := 'False'; ExternalWritable := 'False'} : Bool;   // Service Benutzerdefiniert 1: Bedienerführung angewählt / User-defined service 1: Operator guidance selected
            END_STRUCT;
         END_STRUCT;
         userDefined2 { ExternalAccessible := 'False'; ExternalVisible := 'False'; ExternalWritable := 'False'} : Struct   // Service Benutzerdefiniert 2 / User-defined service 2
            select { ExternalAccessible := 'False'; ExternalVisible := 'False'; ExternalWritable := 'False'} : Bool;   // Service Benutzerdefiniert 2: Anwahl (S) / User-defined service 2: Selection (S)
            deselect { ExternalAccessible := 'False'; ExternalVisible := 'False'; ExternalWritable := 'False'} : Bool;   // Service Benutzerdefiniert 2: Abwahl (S) / User-defined service 2: Deselection (S)
            isActive { ExternalAccessible := 'False'; ExternalVisible := 'False'; ExternalWritable := 'False'} : Bool;   // Service Benutzerdefiniert 2: Aktiv / User-defined service 2: Active
            operatorGuidance { ExternalAccessible := 'False'; ExternalVisible := 'False'; ExternalWritable := 'False'} : Struct   // Service Benutzerdefiniert 2: Bedienerführung / User-defined service 2: Operator guidance
               select { ExternalAccessible := 'False'; ExternalVisible := 'False'; ExternalWritable := 'False'} : Bool;   // Service Benutzerdefiniert 2: Bedienerführung Anwahl (S) / User-defined service 2: Operator guidance selection (S)
               isSelected { ExternalAccessible := 'False'; ExternalVisible := 'False'; ExternalWritable := 'False'} : Bool;   // Service Benutzerdefiniert 2: Bedienerführung angewählt / User-defined service 2: Operator guidance selected
            END_STRUCT;
         END_STRUCT;
         sequenceController { ExternalAccessible := 'False'; ExternalVisible := 'False'; ExternalWritable := 'False'} : Struct   // Ablaufsteuerung (nur auf FG-Ebene) / Sequence control:
            isInitial { ExternalAccessible := 'False'; ExternalVisible := 'False'; ExternalWritable := 'False'} : Bool;   // Ablaufsteuerung ist Initial (Idle / kein Auftrag aktiv / Initialschritt) / Sequence control is initial (idle / no job active / initial step)
            setInitias { ExternalAccessible := 'False'; ExternalVisible := 'False'; ExternalWritable := 'False'} : Struct   // Ablaufstuerung in Initial setzen
               select { ExternalAccessible := 'False'; ExternalVisible := 'False'; ExternalWritable := 'False'} : Bool;   // Ablaufstuerung in Initial setzen: Anwahl (S)
               isSelected { ExternalAccessible := 'False'; ExternalVisible := 'False'; ExternalWritable := 'False'} : Bool;   // Ablaufstuerung in Initial setzen: Angewählt
            END_STRUCT;
            lockForwarding { ExternalAccessible := 'False'; ExternalVisible := 'False'; ExternalWritable := 'False'} : Struct   // Ablaufsteuerung Sperre Schrittweiterschaltung setzen
               select { ExternalAccessible := 'False'; ExternalVisible := 'False'; ExternalWritable := 'False'} : Bool;   // Ablaufsteuerung Sperre Schrittweiterschaltung setzen: Anwahl (S)
               isSelsected { ExternalAccessible := 'False'; ExternalVisible := 'False'; ExternalWritable := 'False'} : Bool;   // Ablaufsteuerung Sperre Schrittweiterschaltung setzen: Angewählt
            END_STRUCT;
         END_STRUCT;
         standstill { ExternalAccessible := 'False'; ExternalVisible := 'False'; ExternalWritable := 'False'} : Struct   // Stillstand / Standstill
            reset { ExternalAccessible := 'False'; ExternalVisible := 'False'; ExternalWritable := 'False'} : Bool;   // Stillstand zurücksetzen (S) / Reset idle state (S)
            isStandingStill { ExternalAccessible := 'False'; ExternalVisible := 'False'; ExternalWritable := 'False'} : Bool;   // im Stillstand / during standstill
         END_STRUCT;
         cyclicClock { ExternalAccessible := 'False'; ExternalVisible := 'False'; ExternalWritable := 'False'} : UInt;   // Zyklustakt (0=Initial, Inkrementiert jeden Zyklus, beginnt bei Überlauf wieder bei 1) / Cycle time (0 = Initial, incremented each cycle, restarts at 1 for overflow
      END_STRUCT;
      faultManagement { ExternalAccessible := 'False'; ExternalVisible := 'False'; ExternalWritable := 'False'} : "typeFaultManagement";   // Störungen / Faults
      summarySignal { ExternalAccessible := 'False'; ExternalVisible := 'False'; ExternalWritable := 'False'} : Struct   // Sammelsignale / Batch signals / Group signals
         cyclicFirstCall { ExternalAccessible := 'False'; ExternalVisible := 'False'; ExternalWritable := 'False'} : Struct   // Sammelsignale Zyklischer Erstaufruf / Group signals cyclical first call
            groupModes { ExternalAccessible := 'False'; ExternalVisible := 'False'; ExternalWritable := 'False'} : Bool;   // Sammelsignale Zyklischer Erstaufruf: Gruppen Modus (wurde für mind. 1 Gruppe durchlaufen) / Group signals cyclical first call: Group mode (run for at least 1 group)
            faults { ExternalAccessible := 'False'; ExternalVisible := 'False'; ExternalWritable := 'False'} : Bool;   // Sammelsignale Zyklischer Erstaufruf: Störungen (wurde für mind. 1 Gruppe durchlaufen) / Group signals cyclical first call: Faults (run for at least 1 group)
            complete { ExternalAccessible := 'False'; ExternalVisible := 'False'; ExternalWritable := 'False'} : Bool;   // Sammelsignale Zyklischer Erstaufruf: Gesamt (wurde für mind. 1 Gruppe durchlaufen) / Group signals cyclical first call: Total (run for at least 1 group)
         END_STRUCT;
         oneUnit { ExternalAccessible := 'False'; ExternalVisible := 'False'; ExternalWritable := 'False'} : Struct   // Sammelsignale: Mindestens ein ... / Group signals: at least one ...
            isPresent { ExternalAccessible := 'False'; ExternalVisible := 'False'; ExternalWritable := 'False'} : Bool;   // Sammelsignal: Mindestens eine Untergruppe vorhanden / Group signal: at least one subgroup present
            groupModes { ExternalAccessible := 'False'; ExternalVisible := 'False'; ExternalWritable := 'False'} : Struct   // Sammelsignale Stations Modus: Mindestens ein ... / Group signals station mode: at least one ...
               isDeactivated { ExternalAccessible := 'False'; ExternalVisible := 'False'; ExternalWritable := 'False'} : Bool;   // Sammelsignale Stations Modus: Mindestens eine Gruppe ist deaktiviert / Group signals station mode: at least one group is deactivated
               isActivated { ExternalAccessible := 'False'; ExternalVisible := 'False'; ExternalWritable := 'False'} : Bool;   // Sammelsignale Stations Modus: Mindestens eine Gruppe ist aktiviert / Group signals station mode: at least one group is activated
               inInterlinkedMode { ExternalAccessible := 'False'; ExternalVisible := 'False'; ExternalWritable := 'False'} : Bool;   // Sammelsignale Stations Modus: Mindestens eine Gruppe ist im "Verketteten Betrieb" / Group signals station mode: at least one group is in "Interlinked mode"
            END_STRUCT;
            baseFunction { ExternalAccessible := 'False'; ExternalVisible := 'False'; ExternalWritable := 'False'} : Struct   // Sammelsignale Grundfunktionen: Mindestens ein ... / Group signals basic functions: at least one ...
               inHomePos { ExternalAccessible := 'False'; ExternalVisible := 'False'; ExternalWritable := 'False'} : Bool;   // Sammelsignale Grundfunktionen: Mindestens eine Gruppe in Grundstellung / Group signals basic functions: at least one group in home position
               toHomePos { ExternalAccessible := 'False'; ExternalVisible := 'False'; ExternalWritable := 'False'} : Struct   // Sammelsignale Grundfunktionen: Mindestens ein "zur Grundstellung"... / Group signals basic functions: At least one "To home position"...
                  isPending { ExternalAccessible := 'False'; ExternalVisible := 'False'; ExternalWritable := 'False'} : Bool;   // Sammelsignale Grundfunktionen: Mindestens ein "zur Grundstellung" steht an (aktiv oder gestoppt) / Group signals basic functions: At least one "To home position" pending (active or stopped)
                  active { ExternalAccessible := 'False'; ExternalVisible := 'False'; ExternalWritable := 'False'} : Bool;   // Sammelsignale Grundfunktionen: Mindestens ein "zur Grundstellung" aktiv / Group signals basic functions: at least one "To home position" active
                  enabled { ExternalAccessible := 'False'; ExternalVisible := 'False'; ExternalWritable := 'False'} : Bool;   // Sammelsignale Grundfunktionen: Mindestens ein "zur Grundstellung" ist freigegeben / Group signals basic functions: At least one "To home position" enabled
               END_STRUCT;
               start { ExternalAccessible := 'False'; ExternalVisible := 'False'; ExternalWritable := 'False'} : Struct   // Sammelsignale Grundfunktionen: Mindestens eine Gruppe Start... / Group signals basic functions: At least one group start...
                  isPending { ExternalAccessible := 'False'; ExternalVisible := 'False'; ExternalWritable := 'False'} : Bool;   // Sammelsignale Grundfunktionen: Mindestens eine Gruppe Start steht an (aktiv oder gestoppt) / Group signals basic functions: At least one group start pending (active or stopped)
                  active { ExternalAccessible := 'False'; ExternalVisible := 'False'; ExternalWritable := 'False'} : Bool;   // Sammelsignale Grundfunktionen: Mindestens eine Gruppe gestartet / Group signals basic functions: at least one group started
                  enabled { ExternalAccessible := 'False'; ExternalVisible := 'False'; ExternalWritable := 'False'} : Bool;   // Sammelsignale Grundfunktionen: Mindestens ein Start freigegeben / Group signals basic functions: at least one start enabled
               END_STRUCT;
               stopped { ExternalAccessible := 'False'; ExternalVisible := 'False'; ExternalWritable := 'False'} : Bool;   // Sammelsignale Grundfunktionen: Mindestens ein Gruppe gestoppt / Group signals basic functions: at least one group stopped
               inReset { ExternalAccessible := 'False'; ExternalVisible := 'False'; ExternalWritable := 'False'} : Bool;   // Sammelsignale Grundfunktionen: Mindestens eine Gruppe in Reset / Group signals basic functions: at least one group in reset
               stopCycleEnd { ExternalAccessible := 'False'; ExternalVisible := 'False'; ExternalWritable := 'False'} : Struct   // Sammelsignale Grundfunktionen: Mindestens ein "Halt nach Taktende"... / Group signals basic functions: At least one "Stop at end of cycle"...
                  active { ExternalAccessible := 'False'; ExternalVisible := 'False'; ExternalWritable := 'False'} : Bool;   // Sammelsignale Grundfunktionen: Mindestens ein "Halt nach Taktende" aktiv / Group signals basic functions: at least one "Stop at end of cycle" active
                  reached { ExternalAccessible := 'False'; ExternalVisible := 'False'; ExternalWritable := 'False'} : Bool;   // Sammelsignale Grundfunktionen: Mindestens ein "Halt nach Taktende" erreicht / Group signals basic functions: at least one "Stop at end of cycle" reached
               END_STRUCT;
               stoppedOrInReset { ExternalAccessible := 'False'; ExternalVisible := 'False'; ExternalWritable := 'False'} : Bool;   // Sammelsignale Grundfunktionen: Mindestens eine Gruppe gestoppt oder im Reset / Group signals basic functions: at least one group stopped or in reset
               singleCycleStep { ExternalAccessible := 'False'; ExternalVisible := 'False'; ExternalWritable := 'False'} : Struct   // Sammelsignale Grundfunktionen Einzelbetrieb/Einzelschritt: Mindestens eine ... / Group signals basic functions single operation/single-step: at least one ...
                  jobSelected { ExternalAccessible := 'False'; ExternalVisible := 'False'; ExternalWritable := 'False'} : Bool;   // Sammelsignale Grundfunktionen Einzelbetrieb/Einzelschritt: Mindestens ein Auftrag angewählt / Group signals basic functions single operation/single-step: at least one job selected
                  homePosStep { ExternalAccessible := 'False'; ExternalVisible := 'False'; ExternalWritable := 'False'} : Struct   // Sammelsignale Grundfunktionen Einzelbetrieb/Einzelschritt: Mindestens ein Grundstellung Einzelschritt ... / Group signals basic functions single operation/single-step: At least one home position single-step ...
                     jobSelected { ExternalAccessible := 'False'; ExternalVisible := 'False'; ExternalWritable := 'False'} : Bool;   // Sammelsignale Grundfunktionen Einzelbetrieb/Einzelschritt: Mindestens ein Grundstellung Einzelschritt angewählt / Group signals basic functions single operation/single-step: At least one home position single-step selected
                     active { ExternalAccessible := 'False'; ExternalVisible := 'False'; ExternalWritable := 'False'} : Bool;   // Sammelsignale Grundfunktionen Einzelbetrieb/Einzelschritt: Mindestens ein Grundstellung Einzelschritt aktiv / Group signals basic functions single operation/single-step: At least one home position single-step active
                  END_STRUCT;
               END_STRUCT;
            END_STRUCT;
            operatingMode { ExternalAccessible := 'False'; ExternalVisible := 'False'; ExternalWritable := 'False'} : Struct   // Sammelsignale Funktionsarten: Mindestens ein ... / Group signals operating modes: at least one ... / Function types group signals: At least one...
               inAutomatic { ExternalAccessible := 'False'; ExternalVisible := 'False'; ExternalWritable := 'False'} : Bool;   // Sammelsignale Funktionsarten: Mindestens eine Gruppe in Automatik / Group signals operating modes: at least one group in automatic mode / Function types group signals: At least one group in Automatic mode
               inSingleCycle { ExternalAccessible := 'False'; ExternalVisible := 'False'; ExternalWritable := 'False'} : Bool;   // Sammelsignale Funktionsarten: Mindestens eine Gruppe in Einzelbetrieb / Group signals operating modes: at least one group in single cycle / Function types group signals: At least one group in Single operation mode
               inSingleStep { ExternalAccessible := 'False'; ExternalVisible := 'False'; ExternalWritable := 'False'} : Bool;   // Sammelsignale Funktionsarten: Mindestens eine Gruppe in Einzelschritt / Group signals operating modes: at least one group in single step / Function types group signals: At least one group in Single-step mode
               inManual { ExternalAccessible := 'False'; ExternalVisible := 'False'; ExternalWritable := 'False'} : Bool;   // Sammelsignale Funktionsarten: Mindestens eine Gruppe in Einrichten / Group signals operating modes: at least one group in setup mode / Function types group signals: At least one group in Setup mode
            END_STRUCT;
            cycleType { ExternalAccessible := 'False'; ExternalVisible := 'False'; ExternalWritable := 'False'} : Struct   // Sammelsignale Taktarten: Mindestens ein ... / Group signals cycle times: at least one ...
               warmUpActive { ExternalAccessible := 'False'; ExternalVisible := 'False'; ExternalWritable := 'False'} : Bool;   // Sammelsignale Taktarten: Mindestens ein Warmfahren aktiv / Group signals cycle times: at least one warm-up cycle active
               runOutActive { ExternalAccessible := 'False'; ExternalVisible := 'False'; ExternalWritable := 'False'} : Bool;   // Sammelsignale Taktarten: Mindestens ein Leerfahren / Group signals cycle times: at least one runout mode
               withoutPartActive { ExternalAccessible := 'False'; ExternalVisible := 'False'; ExternalWritable := 'False'} : Bool;   // Sammelsignale Taktarten: Mindestens ein "Fahren ohne Werkstück" aktiv / Group signals cycle times: at least one "Traverse without part" active
               userDefined1Active { ExternalAccessible := 'False'; ExternalVisible := 'False'; ExternalWritable := 'False'} : Bool;   // Sammelsignale Taktarten: Mindestens ein "Benutzerdefinier 1" aktiv / Group signals cycle types: At least one "User-defined 1" active
               userDefined2Active { ExternalAccessible := 'False'; ExternalVisible := 'False'; ExternalWritable := 'False'} : Bool;   // Sammelsignale Taktarten: Mindestens ein "Benutzerdefinier 2" aktiv / Group signals cycle types: At least one "User-defined 2" active
            END_STRUCT;
            specialSignal { ExternalAccessible := 'False'; ExternalVisible := 'False'; ExternalWritable := 'False'} : Struct   // Sammelsignale Sondersignale: Mindestens ein ... / Group signals special signals: at least one ...
               empty { ExternalAccessible := 'False'; ExternalVisible := 'False'; ExternalWritable := 'False'} : Bool;   // Sammelsignale Sondersignale: Mindestens eine Gruppe ist leer / Group signals special functions: at least one group is empty
               standstill { ExternalAccessible := 'False'; ExternalVisible := 'False'; ExternalWritable := 'False'} : Bool;   // Sammelsignale Sondersignale: Mindestens eine Gruppe im Stillstand / Group signals special signals: At least one group in idle state
               serviceModeActive { ExternalAccessible := 'False'; ExternalVisible := 'False'; ExternalWritable := 'False'} : Bool;   // Sammelsignale Sondersignale: Mindestens eine Gruppe im Servicemodus / Group signals special functions: at least one group in service mode
               stoppedOrInReset { ExternalAccessible := 'False'; ExternalVisible := 'False'; ExternalWritable := 'False'} : Bool;   // Sammelsignale Sondersignale: Mindestens eine Gruppe gestoppt oder im Reset / Group signals special functions: at least one group stopped or in reset
               userDefined1Active { ExternalAccessible := 'False'; ExternalVisible := 'False'; ExternalWritable := 'False'} : Bool;   // Sammelsignale Sondersignale: Mindestens ein "Benutzerdefinier 1" aktiv / Group signals special signals: At least one "User-defined 1" active
               userDefined2Active { ExternalAccessible := 'False'; ExternalVisible := 'False'; ExternalWritable := 'False'} : Bool;   // Sammelsignale Sondersignale: Mindestens ein "Benutzerdefinier 2" aktiv / Group signals special signals: At least one "User-defined 2" active
            END_STRUCT;
            displays { ExternalAccessible := 'False'; ExternalVisible := 'False'; ExternalWritable := 'False'} : Struct   // Sammelsignale Anzeigen: Mindestens ein ... / Group signals displays: at least one ...
               homePos { ExternalAccessible := 'False'; ExternalVisible := 'False'; ExternalWritable := 'False'} : Bool;   // Sammelsignale Anzeige: Mindestens ein Grundstellung / Group signal display: at least one home position
               start { ExternalAccessible := 'False'; ExternalVisible := 'False'; ExternalWritable := 'False'} : Bool;   // Sammelsignale Anzeige: Mindestens ein Start / Group signal display: at least one start
               stop { ExternalAccessible := 'False'; ExternalVisible := 'False'; ExternalWritable := 'False'} : Bool;   // Sammelsignale Anzeige: Mindestens ein Stop / Group signal display: at least one stop
               reset { ExternalAccessible := 'False'; ExternalVisible := 'False'; ExternalWritable := 'False'} : Bool;   // Sammelsignale Anzeige: Mindestens ein Reset / Group signal display: at least one reset
               stopCycleEnd { ExternalAccessible := 'False'; ExternalVisible := 'False'; ExternalWritable := 'False'} : Bool;   // Sammelsignale Anzeige: Mindestens ein "Halt nach Taktende" / Group signals display: at least one "Stop at end of cycle"
            END_STRUCT;
         END_STRUCT;
         allUnits { ExternalAccessible := 'False'; ExternalVisible := 'False'; ExternalWritable := 'False'} : Struct   // Sammelsignale: Alle ... / Group signals: all ...
            groupModes { ExternalAccessible := 'False'; ExternalVisible := 'False'; ExternalWritable := 'False'} : Struct   // Sammelsignale Stations Modus: Alle ... / Group signals station mode: all ...
               isDeactivated { ExternalAccessible := 'False'; ExternalVisible := 'False'; ExternalWritable := 'False'} : Bool;   // Sammelsignale Stations Modus: Alle Gruppen sind deaktiviert / Group signals station mode: all groups are deactivated
               isActivated { ExternalAccessible := 'False'; ExternalVisible := 'False'; ExternalWritable := 'False'} : Bool;   // Sammelsignale Stations Modus: Alle Gruppen sind aktiviert / Group signals station mode: all groups are activated
               inInterlinkedMode { ExternalAccessible := 'False'; ExternalVisible := 'False'; ExternalWritable := 'False'} : Bool;   // Sammelsignale Stations Modus: Alle Gruppen sind im "Verketteten Betrieb" / Group signals station mode: all groups are in "Interlinked mode"
            END_STRUCT;
            baseFunction { ExternalAccessible := 'False'; ExternalVisible := 'False'; ExternalWritable := 'False'} : Struct   // Sammelsignale Grundfunktionen: Alle ... / Group signals basic functions: all ...
               inHomePos { ExternalAccessible := 'False'; ExternalVisible := 'False'; ExternalWritable := 'False'} : Bool;   // Sammelsignale Grundfunktionen: Alle Gruppen in Grundstellung / Group signals basic functions: all groups in home position
               toHomePos { ExternalAccessible := 'False'; ExternalVisible := 'False'; ExternalWritable := 'False'} : Struct   // Sammelsignale Grundfunktionen: Alle Gruppen "zur Grundstellung"... / Group signals basic functions: All groups to home position...
                  isPending { ExternalAccessible := 'False'; ExternalVisible := 'False'; ExternalWritable := 'False'} : Bool;   // Sammelsignale Grundfunktionen: Alle Gruppen "zur Grundstellung" steht an (aktiv oder gestoppt) / Group signals basic functions: All groups "To home position" pending (active or stopped)
                  active { ExternalAccessible := 'False'; ExternalVisible := 'False'; ExternalWritable := 'False'} : Bool;   // Sammelsignale Grundfunktionen: Alle Gruppen "zur Grundstellung" aktiv / Group signals basic functions: All groups "To home position" active
                  enabled { ExternalAccessible := 'False'; ExternalVisible := 'False'; ExternalWritable := 'False'} : Bool;   // Sammelsignale Grundfunktionen: Alle Gruppen "zur Grundstellung" ist freigegeben / Group signals basic functions: All groups "To home position" enabled
               END_STRUCT;
               start { ExternalAccessible := 'False'; ExternalVisible := 'False'; ExternalWritable := 'False'} : Struct   // Sammelsignale Grundfunktionen: Alle Gruppen Start... / Group signals basic functions: All groups start...
                  isPending { ExternalAccessible := 'False'; ExternalVisible := 'False'; ExternalWritable := 'False'} : Bool;   // Sammelsignale Grundfunktionen: Alle Gruppen Start steht an (aktiv oder gestoppt) / Group signals basic functions: All groups start pending (active or stopped)
                  active { ExternalAccessible := 'False'; ExternalVisible := 'False'; ExternalWritable := 'False'} : Bool;   // Sammelsignale Grundfunktionen: Alle Gruppen gestartet / Group signals basic functions: All groups started
                  enabled { ExternalAccessible := 'False'; ExternalVisible := 'False'; ExternalWritable := 'False'} : Bool;   // Sammelsignale Grundfunktionen: Alle Gruppen Start freigegeben / Group signals basic functions: all groups start enabled
               END_STRUCT;
               stopped { ExternalAccessible := 'False'; ExternalVisible := 'False'; ExternalWritable := 'False'} : Bool;   // Sammelsignale Grundfunktionen: Alle Gruppen gestoppt / Group signals basic functions: all groups stopped
               inReset { ExternalAccessible := 'False'; ExternalVisible := 'False'; ExternalWritable := 'False'} : Bool;   // Sammelsignale Grundfunktionen: Alle Gruppen im Reset / Group signals basic functions: all groups in reset
               stopCycleEnd { ExternalAccessible := 'False'; ExternalVisible := 'False'; ExternalWritable := 'False'} : Struct   // Sammelsignale Grundfunktionen: Alle Gruppen "Halt nach Taktende"... / Group signals basic functions: All groups "Stop at end of cycle"...
                  active { ExternalAccessible := 'False'; ExternalVisible := 'False'; ExternalWritable := 'False'} : Bool;   // Sammelsignale Grundfunktionen: Alle Gruppen "Halt nach Taktende" aktiv / Group signals basic functions: all groups "Stop at end of cycle" active
                  reached { ExternalAccessible := 'False'; ExternalVisible := 'False'; ExternalWritable := 'False'} : Bool;   // Sammelsignale Grundfunktionen: Alle Gruppen "Halt nach Taktende" erreicht / Group signals basic functions: all groups "Stop at end of cycle" reached
               END_STRUCT;
               stoppedOrInReset { ExternalAccessible := 'False'; ExternalVisible := 'False'; ExternalWritable := 'False'} : Bool;   // Sammelsignale Grundfunktionen: Alle Gruppen gestoppt oder im Reset / Group signals basic functions: all groups stopped or in reset
               singleCycleStep { ExternalAccessible := 'False'; ExternalVisible := 'False'; ExternalWritable := 'False'} : Struct   // Sammelsignale Grundfunktionen Einzelbetrieb/Einzelschritt: Alle Gruppen ... / Group signals basic functions single operation/single-step: all groups ...
                  jobSelected { ExternalAccessible := 'False'; ExternalVisible := 'False'; ExternalWritable := 'False'} : Bool;   // Sammelsignale Grundfunktionen Einzelbetrieb/Einzelschritt: Alle Gruppen Auftrag angewählt / Group signals basic functions single operation/single-step: all groups job selected
                  homePosStep { ExternalAccessible := 'False'; ExternalVisible := 'False'; ExternalWritable := 'False'} : Struct   // Sammelsignale Grundfunktionen Einzelbetrieb/Einzelschritt: Alle Gruppen Grundstellung Einzelschritt ... / Group signals basic functions single operation/single-step: All groups home position single-step ...
                     jobSelected { ExternalAccessible := 'False'; ExternalVisible := 'False'; ExternalWritable := 'False'} : Bool;   // Sammelsignale Grundfunktionen Einzelbetrieb/Einzelschritt: Alle Gruppen Grundstellung Einzelschritt angewählt / Group signals basic functions single operation/single-step: All groups home position single-step selected
                     active { ExternalAccessible := 'False'; ExternalVisible := 'False'; ExternalWritable := 'False'} : Bool;   // Sammelsignale Grundfunktionen Einzelbetrieb/Einzelschritt: Alle Gruppen Grundstellung Einzelschritt aktiv / Group signals basic functions single operation/single-step: All groups home position single-step active
                  END_STRUCT;
               END_STRUCT;
            END_STRUCT;
            operatingMode { ExternalAccessible := 'False'; ExternalVisible := 'False'; ExternalWritable := 'False'} : Struct   // Sammelsignale Funktionsarten: Alle ... / Group signals operating modes: all ... / Function types group signals: All ...
               inAutomatic { ExternalAccessible := 'False'; ExternalVisible := 'False'; ExternalWritable := 'False'} : Bool;   // Sammelsignale Funktionsarten: Alle Gruppen in Automatik / Group signals operating modes: all groups in automatic mode / Function types group signals: All groups in Automatic mode
               inSingleCycle { ExternalAccessible := 'False'; ExternalVisible := 'False'; ExternalWritable := 'False'} : Bool;   // Sammelsignale Funktionsarten: Alle Gruppen in Einzelbetrieb / Group signals operating modes: all groups in single cycle / Function types group signals: All groups in Single operation mode
               inSingleStep { ExternalAccessible := 'False'; ExternalVisible := 'False'; ExternalWritable := 'False'} : Bool;   // Sammelsignale Funktionsarten: Alle Gruppen in Einzelschritt / Group signals operating modes: all groups in single step / Function types group signals: All groups in Single-step mode
               inManual { ExternalAccessible := 'False'; ExternalVisible := 'False'; ExternalWritable := 'False'} : Bool;   // Sammelsignale Funktionsarten: Alle Gruppen in Einrichten / Group signals operating modes: all groups in setup mode / Function types group signals: All groups in Setup mode
            END_STRUCT;
            cycleType { ExternalAccessible := 'False'; ExternalVisible := 'False'; ExternalWritable := 'False'} : Struct   // Sammelsignale Taktarten: Alle ... / Group signals cycle times: all ...
               warmUpActive { ExternalAccessible := 'False'; ExternalVisible := 'False'; ExternalWritable := 'False'} : Bool;   // Sammelsignale Taktarten: Alle Gruppen Warmfahren aktiv / Group signals cycle times: all groups warm-up cycle active
               runOutActive { ExternalAccessible := 'False'; ExternalVisible := 'False'; ExternalWritable := 'False'} : Bool;   // Sammelsignale Taktarten: Alle Gruppen Leerfahren aktiv / Group signals cycle times: all groups runout mode active
               withoutPartActive { ExternalAccessible := 'False'; ExternalVisible := 'False'; ExternalWritable := 'False'} : Bool;   // Sammelsignale Taktarten: Alle Gruppen "Fahren ohne Werkstück" aktiv / Group signals cycle times: all groups "Traverse without part" active
               userDefined1Active { ExternalAccessible := 'False'; ExternalVisible := 'False'; ExternalWritable := 'False'} : Bool;   // Sammelsignale Taktarten: Alle Gruppen "Reserve1" aktiv / Group signals cycle types: All groups "Reserve 1" active
               userDefined2Active { ExternalAccessible := 'False'; ExternalVisible := 'False'; ExternalWritable := 'False'} : Bool;   // Sammelsignale Taktarten: Alle Gruppen "Reserve2" aktiv / Group signals cycle types: All groups "Reserve 2" active
            END_STRUCT;
            specialSignal { ExternalAccessible := 'False'; ExternalVisible := 'False'; ExternalWritable := 'False'} : Struct   // Sammelsignale Sondersignale: Alle ... / Group signals special signals: all ...
               empty { ExternalAccessible := 'False'; ExternalVisible := 'False'; ExternalWritable := 'False'} : Bool;   // Sammelsignale Sondersignale: Alle Gruppen leer / Group signals special signals: all groups empty
               standstill { ExternalAccessible := 'False'; ExternalVisible := 'False'; ExternalWritable := 'False'} : Bool;   // Sammelsignale Sondersignale: Alle Gruppen im Stillstand / Group signals special signals: All groups in idle state
               serviceModeActive { ExternalAccessible := 'False'; ExternalVisible := 'False'; ExternalWritable := 'False'} : Bool;   // Sammelsignale Sondersignale: Alle Gruppen im Servicemodus / Group signals special signals: all groups in service mode
               userDefined1Active { ExternalAccessible := 'False'; ExternalVisible := 'False'; ExternalWritable := 'False'} : Bool;   // Sammelsignale Sondersignale: Alle Gruppen "Reserve1" aktiv / Group signals special signals: All groups "Reserve 1" active
               userDefined2Active { ExternalAccessible := 'False'; ExternalVisible := 'False'; ExternalWritable := 'False'} : Bool;   // Sammelsignale Sondersignale: Alle Gruppen "Reserve2" aktiv / Group signals special signals: All groups "Reserve 2" active
            END_STRUCT;
            displays { ExternalAccessible := 'False'; ExternalVisible := 'False'; ExternalWritable := 'False'} : Struct   // Sammelsignale Anzeigen: Alle ... / Group signals displays: all ...
               homePos { ExternalAccessible := 'False'; ExternalVisible := 'False'; ExternalWritable := 'False'} : Bool;   // Sammelsignale Anzeige: Alle Grundstellung / Group signal display: all home position
               start { ExternalAccessible := 'False'; ExternalVisible := 'False'; ExternalWritable := 'False'} : Bool;   // Sammelsignale Anzeige: Alle Start / Group signal display: all start
               stop { ExternalAccessible := 'False'; ExternalVisible := 'False'; ExternalWritable := 'False'} : Bool;   // Sammelsignale Anzeige: Alle Stop / Group signal display: all stop
               reset { ExternalAccessible := 'False'; ExternalVisible := 'False'; ExternalWritable := 'False'} : Bool;   // Sammelsignale Anzeige: Alle Reset / Group signal display: all reset
               stopCycleEnd { ExternalAccessible := 'False'; ExternalVisible := 'False'; ExternalWritable := 'False'} : Bool;   // Sammelsignale Anzeige: Alle "Halt nach Taktende" / Group signals display: all "Stop at end of cycle"
            END_STRUCT;
         END_STRUCT;
         diagnostic { ExternalAccessible := 'False'; ExternalVisible := 'False'; ExternalWritable := 'False'} : Struct   // Sammelsignale Diagnose / Group signals diagnostics
            faultGeneral { ExternalAccessible := 'False'; ExternalVisible := 'False'; ExternalWritable := 'False'} : Bool;   // Sammelsignale Diagnose: Störung steht an / Group signals diagnostics fault pending
            faultMachineOff { ExternalAccessible := 'False'; ExternalVisible := 'False'; ExternalWritable := 'False'} : Bool;   // Sammelsignale Diagnose: Störung sofort halt mit Maschine aus steht an / Group signals diagnostics: fault immediate stop with machine off pending
            faultActive { ExternalAccessible := 'False'; ExternalVisible := 'False'; ExternalWritable := 'False'} : Bool;   // Sammelsignal Diagnose: Störung ist aktiv / Group signal diagnosis: Fault active
            messageGeneral { ExternalAccessible := 'False'; ExternalVisible := 'False'; ExternalWritable := 'False'} : Bool;   // Sammelsignale Diagnose: Meldung / Group signals diagnostics: message
            messageOperatorCall { ExternalAccessible := 'False'; ExternalVisible := 'False'; ExternalWritable := 'False'} : Bool;   // Sammelsignale Diagnose: Meldung mit Bedienerruf steht an / Group signals diagnostics: message with operator call pending
         END_STRUCT;
         generalEnables { ExternalAccessible := 'False'; ExternalVisible := 'False'; ExternalWritable := 'False'} : Struct   // Generelle Freigaben / General enables
            enterSafeArea { ExternalAccessible := 'False'; ExternalVisible := 'False'; ExternalWritable := 'False'} : Bool;   // Freigabe Zugang Schutzbereich gesamt steht an / Enable for access all guarded area pending
         END_STRUCT;
      END_STRUCT;
      mso { ExternalAccessible := 'False'; ExternalVisible := 'False'; ExternalWritable := 'False'} : "typeMSOs";   // MSO
      masterSlaveFg { ExternalAccessible := 'False'; ExternalVisible := 'False'; ExternalWritable := 'False'} : Struct   // Master/Slave Fg / Master/slave Fg
         isSlave { ExternalAccessible := 'False'; ExternalVisible := 'False'; ExternalWritable := 'False'} : Bool;   // Gruppe in Slave-Modus (S) / Group in slave mode (S)
         masterFg { ExternalAccessible := 'False'; ExternalVisible := 'False'; ExternalWritable := 'False'} : Struct   // Master FG
            "name" { ExternalAccessible := 'False'; ExternalVisible := 'False'; ExternalWritable := 'False'} : WString["GRP_JOB_NAME_SIZE"];   // Master FG: Bezeichnung / Master FG: Designation
            inHomePosition { ExternalAccessible := 'False'; ExternalVisible := 'False'; ExternalWritable := 'False'} : Bool;   // Master FG befindet sich in Grundstellung (R) / Master FG in home position (R)
            inStopAtCycleEnd { ExternalAccessible := 'False'; ExternalVisible := 'False'; ExternalWritable := 'False'} : Bool;   // Master FG hat Halt nach Taktende erreicht (R) / Master FG stop at end of cycle reached (R)
         END_STRUCT;
      END_STRUCT;
   END_STRUCT;
   // // specialSignal.userLevel.userLevelBitByBit : Benutzerlevel: Aktives Benutzerlevel Bitweise / User level: active user level bit by bit
   // // specialSignal.userLevel.userLevel : Benutzerlevel: Aktives Benutzerlevel / User level: active user level
   // // specialSignal.userLevel.userLevelChanged : Benutzerlevel: Aktives Benutzerlevel gewechselt / User level: active user level changed
   // // faultManagement.selectAckFault : Anwahl Störung quittieren (S) / Selection: acknowledge fault (S)
   // // faultManagement.ackFault : Störung quittieren / Acknowledge fault
   // // faultManagement.faultGeneral : Generelle Störung steht an / General fault pending
   // // faultManagement.faultInstantStop : Störung sofort Halt steht an / Fault immediate stop pending
   // // faultManagement.faultMachineOut : Störung sofort Halt und Maschine Aus steht an / Fault immediate stop and machine off pending
   // // faultManagement.faultInCycleEnd : Störung Halt nach Taktende steht an / Fault stop at end of cycle pending
   // // faultManagement.faultNoStop : Störung ohne Stop steht an / Fault without stop pending
   // // faultManagement.faultActive : Störung ist aktiv (aus eigener oder übergeordeten Gruppen) / Fault is active (from separate or superordinate groups)
   // // faultManagement.messageGeneral : Meldung steht an / Message pending
   // // faultManagement.messageOperatorCall : Meldung mit Bedienerruf steht an / Message with operator call pending
   // // faultManagement.selectInstantStop : Anwahl sofort Halt bei Störung (S) / Selection immediate stop in case of fault (S)
   // // faultManagement.selectStopCycleEnd : Anwahl Halt nach Taktende bei Störung (S) / Selection stop at end of cycle in case of fault (S)
   // // faultManagement.faultInstantStopByParent : Störung sofort Halt von übergeordneter Baugruppe / Fault immediate stop from superordinate assembly
   // // faultManagement.faultInCycleEndByParent : Störung Halt nach Taktende von übergeordneter Baugruppe / Fault stop at end of cycle from the superordinate assembly
   // // mso.activeMSO2 : MSO: Betriebsart 2 aktiv + Zustimmtaster gedrückt / MSO: Operating mode 2 active + enabling button pressed
   // // mso.activeMSO3 : MSO: Betriebsart 3 aktiv + Zustimmtaster gedrückt / MSO: Operating mode 3 active + enabling button pressed
   // // mso.selectedMSO2 : MSO: Betriebsart 2 angewählt / MSO: Operating mode 2 selected
   // // mso.selectedMSO3 : MSO: Betriebsart 3 angewählt / MSO: Operating mode 3 selected
END_TYPE

TYPE "typeFgControlGeneral"
TITLE = Control interface / Steuershnittstelle
// Control interface [V 01.02 | Kernel_V2] / Steuershnittstelle [V 01.02 | Kernel_V2]
// stored: IsFailsafeCompliant false
   STRUCT
      homePosConditions : Bool;   // Grundstellungsbedingungen / Home position conditions
      waitingPositionStep : Bool;   // Warteschritt / Waiting step
      homePostionStep : Bool := TRUE;   // Grundstellungsschritt akitv / Home position step active
      withoutExecutionStep : Bool;   // Schritt ohne Bewegung / Step without movement
      jobNumber : Int;   // Auftragsnummer / Job number
      activeJobNumber : Int := -1;   // Aktive Auftragsnummer von Ablaufsteuerung / Active job number from sequence control
      seqNumber : Int;   // Schrittnummer / Step number
      internalSignals : Struct   // Steuersignale (nur für internen gebrauch!) ... / Control signals (for internal use only!) ...
         startDelayed : Struct   // Verzögerte Startsingale... / Delayed start signals...
            inExecution : Bool;   // Start aktiv verzögert / Start active delayed
            inExecutionPulse : Bool;   // Start aktiv Impuls verzögert / Start active impulse delayed
         END_STRUCT;
      END_STRUCT;
   END_STRUCT;
END_TYPE

TYPE "typeFgLogEntry"
TITLE = FG log entry / FG-Log Eintrag
// FG log entry [V 01.00 | Kernel_V2] / FG-Log Eintrag [V 01.00 | Kernel_V2]
// stored: IsFailsafeCompliant false
   STRUCT
      area { ExternalAccessible := 'False'; ExternalVisible := 'False'; ExternalWritable := 'False'} : Byte;   // 16#FF Header | 16#01 Log Entry | 16#00 Empty
      pointerOrEventId { ExternalAccessible := 'False'; ExternalVisible := 'False'; ExternalWritable := 'False'} : DWord;   // Area = 16#00: Pointer auf letzten Eintrag | Area = 16#01: Event-ID / Area = 16#00: Pointer at last entry | Area = 16#01: Event ID
      opMode { ExternalAccessible := 'False'; ExternalVisible := 'False'; ExternalWritable := 'False'} : Byte;   // 16#01 Automatic | 16#02 SingleCycle | 16#04 SingleStep | 16#08 Manual | 16#10 MSO 2 | 16#20 MSO 3 | 16#40 MSO GROB
      baseFunction { ExternalAccessible := 'False'; ExternalVisible := 'False'; ExternalWritable := 'False'} : Byte;   // 16#00 Reset | 16#01 Stop is active | 16#02 Start is active | 16#03 Start is stopped | 16#04 HomePos active | 16#05 HomePos is stopped | 16#10 in HomePos | 16#20 Stop at cycle active
      cycleType { ExternalAccessible := 'False'; ExternalVisible := 'False'; ExternalWritable := 'False'} : Byte;   // 16#01 Empying Mode | 16#02 Dry Run | 16#04 WarmUp | 16#08 UserDef 1 | 16#10 UserDef 2
      groupMode { ExternalAccessible := 'False'; ExternalVisible := 'False'; ExternalWritable := 'False'} : Byte;   // 16#01 Group active | 16#02 Group in Interlinked Mode | 16#04 Interlock Bypass Mode
      actJobNum { ExternalAccessible := 'False'; ExternalVisible := 'False'; ExternalWritable := 'False'} : Int;   // Aktive Auftragsnummer / Active job number
      sequStepNum { ExternalAccessible := 'False'; ExternalVisible := 'False'; ExternalWritable := 'False'} : Int;   // Ablauf Schrittnummer / Sequence step number
      timeStamp { ExternalAccessible := 'False'; ExternalVisible := 'False'; ExternalWritable := 'False'} : Date_And_Time;   // Zeitstempel / Time stamp
   END_STRUCT;
END_TYPE

TYPE "typeHmiCounter"
TITLE = HMI part counter / HMI Stückzähler
// HMI Stückzähler [V 01.01 | Kernel_V2]
// stored: IsFailsafeCompliant false
   STRUCT
      count : Bool;   // Zählimpuls / Count pulse
      countValue : Byte;   // Anzahl der zu zählenden Gesamtteile (Gut- und Schlechtteile) / Number of parts that are counted
      countValueBad : Byte;   // Anzahl der zu zählenden Schlechtteile / Number of parts that are counted
      typIndex : Word;   // Index des Werkstücktyps, der gezählt werden soll. Bei Wert = 0 wird nur der Gesamtstückzähler berücksichtigt. Werte kleiner 0 haben eine Fehlermeldung zur Folge.
   END_STRUCT;
END_TYPE

TYPE "typeHmiDataSave"
TITLE = Save HMI data / HMI Daten sichern
// HMI Data backup [V 01.00 | Kernel_V2] / HMI Daten sichern [V 01.00 | Kernel_V2]
// stored: IsFailsafeCompliant false
   STRUCT
      saved : Bool;   // Daten gesichert / Data backed up
      resaved : Bool;   // Daten rückgesichert / Data backed up
      resavedComplete : Bool;   // Daten mit Aktualwerten rückgesichert / Data with actual value backed up
      resavedTrig : Bool;   // Daten rückgesichert Trigger / Data backed up trigger
      saveActive : Bool;   // Daten sichern aktiv / Save data active
      resaveActive : Bool;   // Daten rücksichern aktiv / Backup data active
      resaveCompleteActive : Bool;   // Daten rücksichern mit Aktualwerten aktiv / Backup data with actual values active
      backupBufferInitial : Bool;   // Daten Backup-Puffer ist initial / Data backup buffer initialized
      notUpToDate : Bool;   // Daten Sicherung ist nicht aktuell / Data backup not up to date
   END_STRUCT;
END_TYPE

TYPE "typeHmiManualGroup"
TITLE = HMI setup groups / HMI Einricht Gruppen
// HMI Setup groups [V 01.00 | Kernel_V2] / HMI Einricht Gruppen [V 01.00 | Kernel_V2]
// stored: IsFailsafeCompliant false
   STRUCT
      selectedGroup : Array[1..30] of Bool;   // Gruppe Handbedienbild / Group manual operating screen
      manualButtonRight : Bool;   // rechte Taste gedrückt / Right key pressed
      manualButtonLeft : Bool;   // linke Taste gedrückt / Left key pressed
   END_STRUCT;
END_TYPE

TYPE "typeHmiOperatorPrompt"
// stored: IsFailsafeCompliant false
   STRUCT
      promt : Struct
         prompt1 : Bool;   // Bitte warten
         prompt2 : Bool;   // -
         prompt3 : Bool;   // -
         prompt4 : Bool;   // -
         prompt5 : Bool;   // Schweißmaskenwechsel - Montagehilfe nicht vorhanden
         prompt6 : Bool;   // Schweißmaskenwechsel - Schutztüre nicht geöffnet
         prompt7 : Bool;   // Schweißmaskenwechsel - DMC-Code Schweißmaske nicht korrekt
         prompt8 : Bool;   // Leistung ausschalten --> 'Start Aus'
         prompt9 : Bool;   // -
         prompt10 : Bool;   // Not-Halt Hauptbedienpult aufheben
         prompt11 : Bool;   // Not-Halt Mobile Panel aufheben
         prompt12 : Bool;   // Not-Halt Schutztüre 1 aufheben
         prompt13 : Bool;   // Not-Halt Schutztüre 2 aufheben
         prompt14 : Bool;   // Not-Halt Lasergerät 1 aufheben
         prompt15 : Bool;   // Not-Halt Lasergerät 2 aufheben
         prompt16 : Bool;   // Not-Halt Lasergerät 1 Bedienpult aufheben
         prompt17 : Bool;   // Not-Halt Lasergerät 1 Bedienpult aufheben
         prompt18 : Bool;   // -
         prompt19 : Bool;   // -
         prompt20 : Bool;   // Medien gesamt einschalten
         prompt21 : Bool;   // -
         prompt22 : Bool;   // -
         prompt23 : Bool;   // -
         prompt24 : Bool;   // Schutzeinrichtungen schliessen und verriegeln
         prompt25 : Bool;   // Schutztüre 1 schliessen
         prompt26 : Bool;   // Schutztüre 2 schliessen
         prompt27 : Bool;   // -
         prompt28 : Bool;   // -
         prompt29 : Bool;   // -
         prompt30 : Bool;   // Zustimmbetrieb nicht möglich --> mehr als eine Schutztür offen
         prompt31 : Bool;   // Zustimmtaste drücken
         prompt32 : Bool;   // -
         prompt33 : Bool;   // Leistungsmessgerät in Vorrichtung schieben und sichern
         prompt34 : Bool;   // Leistungsmessgerät und Beam-Watch in Vorrichtung schieben und sichern
         prompt35 : Bool;   // Opferblech Laser 1 ist verschlissen --> Wechseln
         prompt36 : Bool;   // Opferblech Laser 2 ist verschlissen --> Wechseln
         prompt37 : Bool;   // -
         prompt38 : Bool;   // -
         prompt39 : Bool;   // Leistung einschalten --> 'Start Ein'
         prompt40 : Bool;   // Start nicht möglich --> 'zur Grundstellung'
         prompt41 : Bool;   // Station starten --> 'Start'
         prompt42 : Bool;   // -
         prompt43 : Bool;   // -
         prompt44 : Bool;   // maximal eine Schutzeinrichtung öffnen/unterbrechen
         prompt45 : Bool;   // -
         prompt46 : Bool;   // -
         prompt47 : Bool;   // -
         prompt48 : Bool;   // -
         prompt49 : Bool;   // Start nicht möglich --> 'zur Grundstellung'
         prompt50 : Bool;   // Station starten --> 'Start'
         prompt51 : Bool;   // -
         prompt52 : Bool;   // -
         prompt53 : Bool;   // -
         prompt54 : Bool;   // -
         prompt55 : Bool;   // -
         prompt56 : Bool;   // -
         prompt57 : Bool;   // -
         prompt58 : Bool;   // -
         prompt59 : Bool;   // -
         prompt60 : Bool;   // -
         prompt61 : Bool;   // -
         prompt62 : Bool;   // -
         prompt63 : Bool;   // -
         prompt64 : Bool;   // Typwechsel quittieren
         prompt65 : Bool;   // SPR-Check ausführen und quittieren
         prompt66 : Bool;   // Missbrauchstest Stopp 1 erforderlich
         prompt67 : Bool;   // Missbrauchstest Stopp 2 erforderlich
         prompt68 : Bool;   // Missbrauchstest Stopp 3 erforderlich
         prompt69 : Bool;   // Missbrauchstest Stopp 4 erforderlich
         prompt70 : Bool;   // Missbrauchstest inaktiv (Zeit- und Stückzahlsteuerung deaktiviert)
         prompt71 : Bool;   // -
         prompt72 : Bool;   // -
         prompt73 : Bool;   // -
         prompt74 : Bool;   // Daten: Sicherungspuffer ist initial -> Daten sichern oder rücksichern!
         prompt75 : Bool;   // Daten Sicherung nicht aktuell
         prompt76 : Bool;   // Verschleißzähler: Sicherung ist initial -> Daten sichern oder rücksichern
         prompt77 : Bool;   // Verschleißzählerdaten nicht aktuell
         prompt78 : Bool;   // -
         prompt79 : Bool;   // -
         prompt80 : Bool;   // -
         prompt81 : Bool;   // -
         prompt82 : Bool;   // -
         prompt83 : Bool;   // -
         prompt84 : Bool;   // -
         prompt85 : Bool;   // -
         prompt86 : Bool;   // -
         prompt87 : Bool;   // -
         prompt88 : Bool;   // -
         prompt89 : Bool;   // -
         prompt90 : Bool;   // -
         prompt91 : Bool;   // -
         prompt92 : Bool;   // -
         prompt93 : Bool;   // -
         prompt94 : Bool;   // -
         prompt95 : Bool;   // -
         prompt96 : Bool;   // -
         prompt97 : Bool;   // -
         prompt98 : Bool;   // -
         prompt99 : Bool;   // -
         prompt100 : Bool;   // -
         prompt101 : Bool;   // -
         prompt102 : Bool;   // -
         prompt103 : Bool;   // -
         prompt104 : Bool;   // -
         prompt105 : Bool;   // -
         prompt106 : Bool;   // -
         prompt107 : Bool;   // -
         prompt108 : Bool;   // -
         prompt109 : Bool;   // -
         prompt110 : Bool;   // -
         prompt111 : Bool;   // -
         prompt112 : Bool;   // -
         prompt113 : Bool;   // -
         prompt114 : Bool;   // -
         prompt115 : Bool;   // -
         prompt116 : Bool;   // -
         prompt117 : Bool;   // -
         prompt118 : Bool;   // -
         prompt119 : Bool;   // -
         prompt120 : Bool;   // -
         prompt121 : Bool;   // -
         prompt122 : Bool;   // -
         prompt123 : Bool;   // -
         prompt124 : Bool;   // -
         prompt125 : Bool;   // -
         prompt126 : Bool;   // -
         prompt127 : Bool;   // -
         prompt128 : Bool;   // -
         prompt129 : Bool;   // -
         prompt130 : Bool;   // -
         prompt131 : Bool;   // -
         prompt132 : Bool;   // -
         prompt133 : Bool;   // -
         prompt134 : Bool;   // -
         prompt135 : Bool;   // -
         prompt136 : Bool;   // -
         prompt137 : Bool;   // -
         prompt138 : Bool;   // -
         prompt139 : Bool;   // -
         prompt140 : Bool;   // -
         prompt141 : Bool;   // -
         prompt142 : Bool;   // -
         prompt143 : Bool;   // -
         prompt144 : Bool;   // -
         prompt145 : Bool;   // -
         prompt146 : Bool;   // -
         prompt147 : Bool;   // -
         prompt148 : Bool;   // -
         prompt149 : Bool;   // -
         prompt150 : Bool;   // -
         prompt151 : Bool;   // -
         prompt152 : Bool;   // -
         prompt153 : Bool;   // -
         prompt154 : Bool;   // -
         prompt155 : Bool;   // -
         prompt156 : Bool;   // -
         prompt157 : Bool;   // -
         prompt158 : Bool;   // -
         prompt159 : Bool;   // -
         prompt160 : Bool;   // -
      END_STRUCT;
   END_STRUCT;
END_TYPE

TYPE "typeHmiScreen"
TITLE = Manual HMI operating screens / HMI Handbedienbilder
// HMI manual operation screens [V 01.00 | Kernel_V2] / HMI Handbedienbilder [V 01.00 | Kernel_V2]
// stored: IsFailsafeCompliant false
   STRUCT
      setup : Struct   // Handbedienbild Einrichten / Manual operating screen 'Setup'
         activ : Bool;   // Aktiv / Active
      END_STRUCT;
      powerup : Struct   // Handbedienbild Einschaltbedingung / Manual operating screen 'Switch-on condition'
         activ : Bool;   // Aktiv / Active
      END_STRUCT;
      unit : Struct   // Handbedienbild Einheiten / Manual operating screen 'Units'
         activ : Bool;   // Aktiv / Active
      END_STRUCT;
      nutrunner : Struct   // Handbedienbild Schrauber / Manual operating screen 'Nut runner'
         activ : Bool;   // Aktiv / Active
      END_STRUCT;
      nutrunnerGroup : Struct   // Handbedienbild Schraubergruppen / Manual operating screen 'Nut runner groups'
         activ : Bool;   // Aktiv / Active
      END_STRUCT;
      cycletype : Struct   // Handbedienbild Taktarten / Manual operating screen 'Cycle types'
         activ : Bool;   // Aktiv / Active
      END_STRUCT;
      userDefine : Struct   // Handbedienbild Anwender / Manual operating screen 'User'
         activ : Bool;   // Aktiv / Active
      END_STRUCT;
   END_STRUCT;
END_TYPE

TYPE "typeHmiSelectedRow"
TITLE = HMI selected line / HMI Ausgewählte Zeile
// HMI selected line [V 01.00 | Kernel_V2] / HMI Ausgewählte Zeile [V 01.00 | Kernel_V2]
// stored: IsFailsafeCompliant false
   STRUCT
      selectedRow : Array[1..348] of Bool;   // Angewählte Zeile / selected line
   END_STRUCT;
END_TYPE

TYPE "typeHmiUserManagement"
TITLE = HMI user management / HMI Benutzerverwaltung
// HMI user management [V 01.00 | Kernel_V2] / HMI Benutzerverwaltung [V 01.00 | Kernel_V2]
// stored: IsFailsafeCompliant false
   STRUCT
      activeUserLevel : "typeUserLevel";   // Benutzerlevel / User level
      eks : Struct   // EKS Protection Level / EKS protection level
         protectionLevel : Int;   // Ausgabe der Schutzstufe / Output of protection level
         checksumNok : Bool;   // EKS Checksumme des Schlüssels n.i.O. / EKS check sum of key NOK
         dateNok : Bool;   // EKS Ablaufdatum des Schlüssels n.i.O. / EKS expiry data of key NOK
         costCenterNok : Bool;   // EKS Kostenstelle des Schlüssels n.i.O. / EKs cost center of key NOK
         eksKeyInvalidLess30Days : Bool;   // EKS Schlüssel wird in 30 Tagen ungültig / EKS key will expire in 30 days
         eksAdapterReady : Bool;   // EKS Adapter betriebsbereit / EKS adapter ready for operation
         eksKeyDetected : Bool;   // EKS Schlüssel erkannt / EKS key detected
         operatiorId : Int;   // EKS Operator ID / EKS operator ID
      END_STRUCT;
   END_STRUCT;
END_TYPE

TYPE "typeUserLevel"
TITLE = HMI user levels / HMI Benutzerstufen
// HMI user levels [V 01.00 | Kernel_V2] / HMI Benutzerstufen [V 01.00 | Kernel_V2]
// stored: IsFailsafeCompliant false
   STRUCT
      userLevelBitByBit : Struct   // Aktives Benutzerlevel Bitweise / Active user level bit by bit
         level1 : Bool;   // Benutzerlevel 1 (Admin) / User level 1 (Admin)
         level2 : Bool;   // Benutzerlevel 2 (Hersteller) / User level 2 (Manufacturer)
         level3 : Bool;   // Benutzerlevel 3 (Instandhaltung) / User level 3 (Maintenance)
         level4 : Bool;   // Benutzerlevel 4 (User) / User level 4 (User)
         level5 : Bool;   // Benutzerlevel 5 (Keyswitch 3) / User level 5 (Keyswitch 3)
         level6 : Bool;   // Benutzerlevel 6 (Keyswitch 2) / User level 6 (Keyswitch 2)
         level7 : Bool;   // Benutzerlevel 7 (Keyswicht 1) / User level 7 (Keyswitch 1)
         level8 : Bool;   // Benutzerlevel 8 () / User level 8 ()
      END_STRUCT;
      userLevel : Int;   // Aktives Benutzerlevel / Active user level
      userLevelChanged : Bool;   // Aktives Benutzerlevel gewechselt / Active user level changed
   END_STRUCT;
END_TYPE

TYPE "typeMSOs"
// stored: IsFailsafeCompliant false
   STRUCT
      activeMSO2 : Bool;   // Betriebsart 2 aktiv + Zustimmtaster gedrückt
      activeMSO3 : Bool;   // Betriebsart 3 aktiv + Zustimmtaster gedrückt
      selectedMSO2 : Bool;   // Betriebsart 2 angewählt
      selectedMSO3 : Bool;   // Betriebsart 3 angewählt
   END_STRUCT;
END_TYPE

